{attribute addProperty BoxType "AT2050-0500-0021"}
{attribute addProperty Id "A_0092_AT2020_5250_0018_AT2020_5250AT2020_3DCFC8D064080"}
{attribute addProperty CRC "3054898156"}
{attribute addProperty SizeInBites "640"}
{attribute addProperty SizeInBytes "80"}
TYPE A_0052_AT2050_0500_0021_B6160BEC EXTENDS AT2050_9506A482 :
STRUCT
	{attribute addProperty Name "A_0092_AT2020_5250_0018_AT2020_5250"}
	A_0092_AT2020_5250_0018_AT2020_5250 : AT2020_3DCFC8D0;
END_STRUCT
END_TYPE

(* stored: Version 1.2.0.0, ProductVersion 3.1.4024.9
   DUT A_0052_AT2050_0500_0021_B6160BEC: Id {70969077-9624-4845-a500-cb161075e62a} *)
